TYPE FsT_Ptr : POINTER TO BYTE; END_TYPE

(* stored: Version 1.1.0.1, ProductVersion 3.1.4024.4
   DUT FsT_Ptr: Id {5abc46be-a59f-4cfa-ae5c-14c241a720f9} *)
